PROGRAM PRG_06_ElectricalMonitoring
VAR
	ElectDeviceContOper					: ElectricalDeviceContOper;
	ElectDeviceContOperPostHttp			: HttpPost;
	ElectrDeviceContOper				: ReadMBSentron_PAC1200;
END_VAR

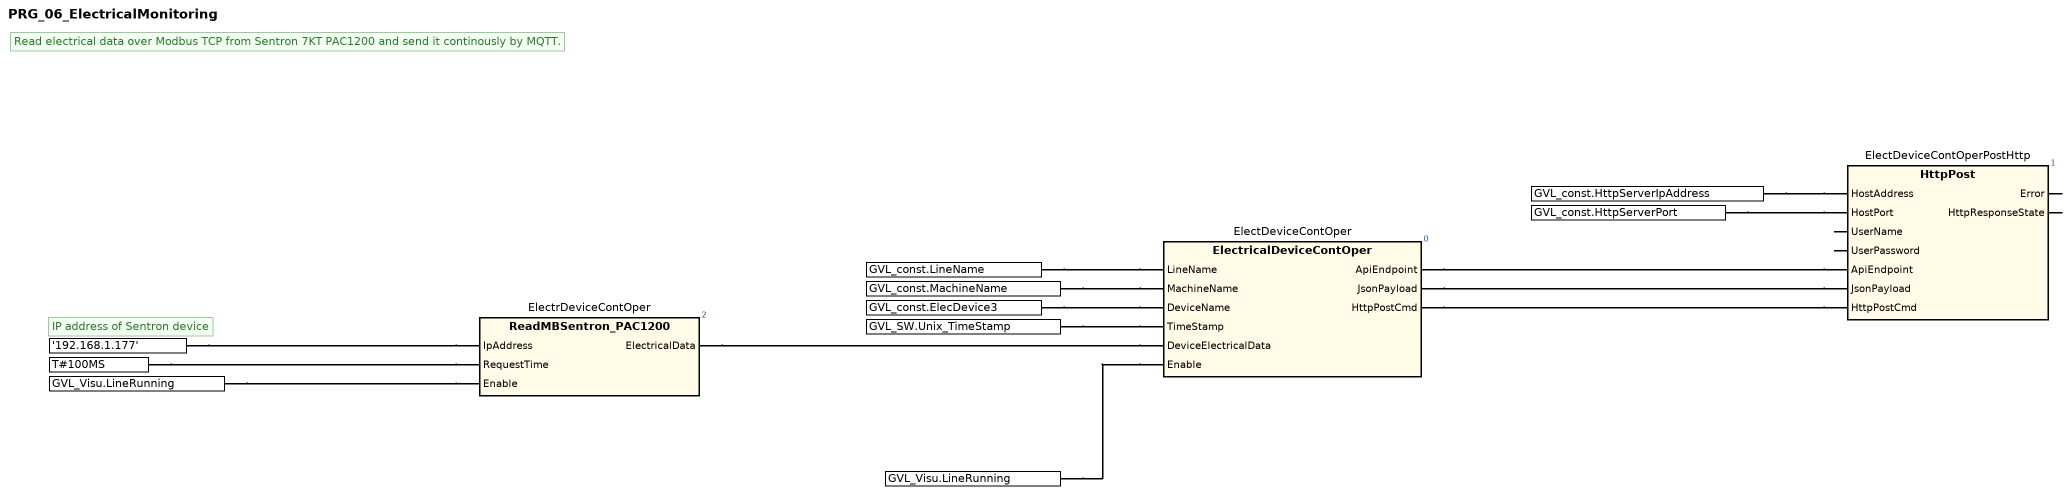
ElectDeviceContOper(
    LineName := GVL_const.LineName,
    MachineName := GVL_const.MachineName,
    DeviceName := GVL_const.ElecDevice3,
    TimeStamp := GVL_SW.Unix_TimeStamp,
    DeviceElectricalData := ElectrDeviceContOper.ElectricalData,
    Enable := GVL_Visu.LineRunning); // ElectricalDeviceContOper
ElectDeviceContOperPostHttp(
    HostAddress := GVL_const.HttpServerIpAddress,
    HostPort := GVL_const.HttpServerPort,
    ApiEndpoint := ElectDeviceContOper.ApiEndpoint,
    JsonPayload := ElectDeviceContOper.JsonPayload,
    HttpPostCmd := ElectDeviceContOper.HttpPostCmd); // HttpPost
// Read electrical data over Modbus TCP from Sentron 7KT PAC1200 and send it continously by MQTT.
// IP address of Sentron device
ElectrDeviceContOper(IpAddress := '192.168.1.177', RequestTime := T#100MS, Enable := GVL_Visu.LineRunning); // ReadMBSentron_PAC1200

END_PROGRAM

(* stored: Version 1.1.0.1, ProductVersion 3.1.4024.15
   POU PRG_06_ElectricalMonitoring: Id {b708dd0b-ad61-45f0-8b7b-5a47f48b89f6}, SpecialFunc None *)
